# EPICS substitutions: dl205/dl205App/Db/depo-plc-write.substitutions
file "depo-plc-write.template" { pattern
 {P	, R			}
 {Depo	, "{PLC:1}Enbl:Write"	}
}
